// LS Electric XG5000 project: 9_3_mini_project
// PLC LSPLC

PROGRAM NewProgram (task: 스캔 프로그램)

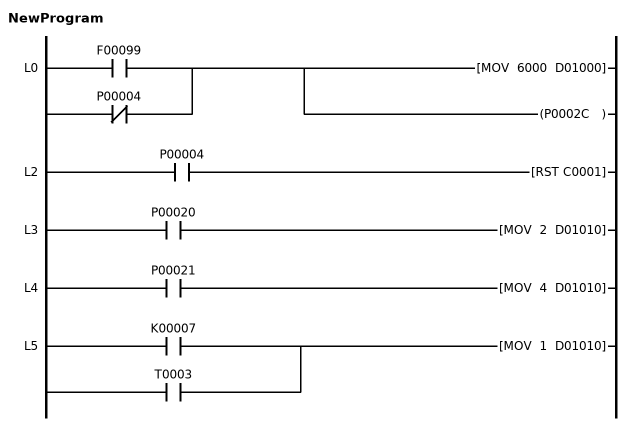
; L0
LOAD      F00099
OR NOT    P00004
MOV       6000 D01000
OUT       P0002C
; L2
LOAD      P00004
RST       C0001
; L3
LOAD      P00020
MOV       2 D01010
; L4
LOAD      P00021
MOV       4 D01010
; L5
LOAD      K00007
OR        T0003
MOV       1 D01010

VARIABLES AND COMMENTS (devices not used above)
P00006	BIT	SEN1
P00007	BIT	SEN2